RoboDK station: MitsubishiWithPython.rdk

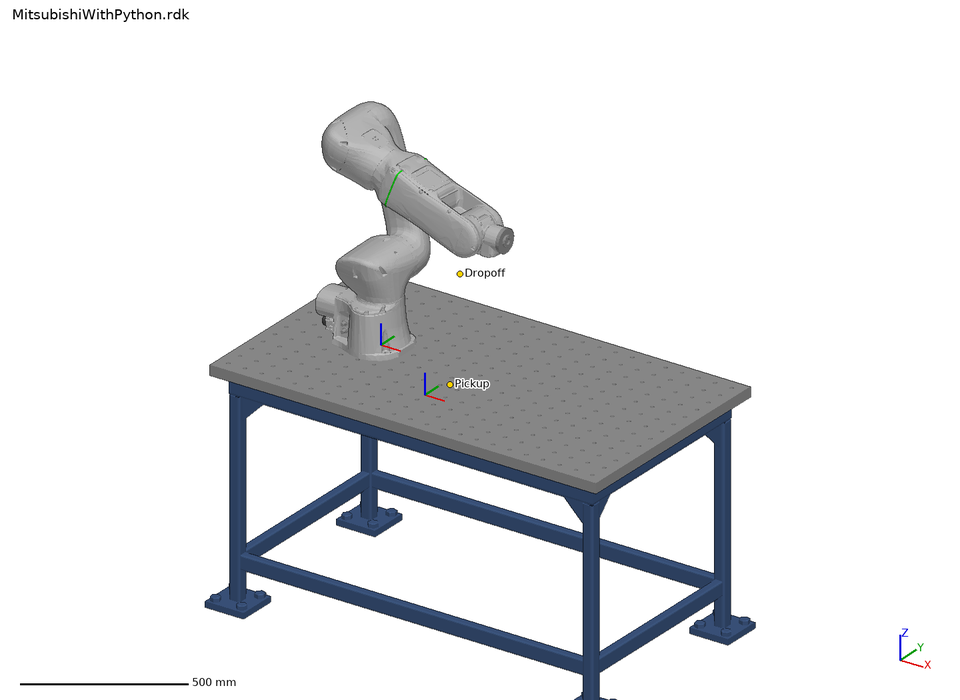
[picture v0: the station drawn from its stored meshes, robots at their saved joint values, targets as dots, program paths as lines]
Station MitsubishiWithPython (saved by RoboDK 5.7.3). Poses are relative to the parent item; angles as X-Y-Z fixed-axis rotations.
  - frame Frame RV-5AS-D at (0, 0, 0) mm
    - robot Mitsubishi RV-5AS-D: 6 axes, payload 5 kg, reach 900 mm, repeatability 0.02 mm, weight 58 kg
        modified DH rows (alpha deg, a mm, theta deg, d mm): 0, 0, 0, 254; -90, 0, -90, 0; 0, 410, -90, 0; -90, 0, 0, 500; 90, 0, 0, 0; -90, 0, 180, 125
        joint limits [-240, -148, -150, -200, -120, -200] to [240, 148, 150, 200, 120, 200]; home [0, 0, 90, 0, 0, 0]; saved at [-1.402, -18.281, 127.838, -4.182, -19.605, 5.574]
  - object Table 1400x800x800mm at (0, 0, 0) mm, size 1420 x 820 x 800 mm, geometry from Table-1400x800x800mm.sld
  - Python program Prog1 (listed below)
  - frame GameFrame at (300, -200, 0) mm
    - target Dropoff (Cartesian target) at (167.45, -58.28, 468.81) mm, rotated rx 90 ry 88.37 rz 90 deg; joints [-37.024, -4.466, 117.289, -62.783, -42.619, 56.684] of Mitsubishi RV-5AS-D
    - target Pickup (Cartesian target) at (71.75, 27.51, 42.52) mm, rotated rx 179.92 ry -4.62 rz -178.08 deg; joints [-24.291, 28.472, 124.985, -183.849, -30.78, 157.175] of Mitsubishi RV-5AS-D

--- Python program Prog1 ---
from robodk.robolink import *  # RoboDK API
from robodk.robomath import *  # RoboDK math utilities

# Initialiser RoboDK API
RDK = Robolink()

# Finn roboten
robot = RDK.Item('', ITEM_TYPE_ROBOT)

if not robot.Valid():
    raise Exception("Ingen robot funnet. Vennligst last inn en robot i RoboDK.")

# Finn targets
pickup_target = RDK.Item("Pickup", ITEM_TYPE_TARGET)
dropoff_target = RDK.Item("Dropoff", ITEM_TYPE_TARGET)

if not pickup_target.Valid() or not dropoff_target.Valid():
    raise Exception("Pickup eller Dropoff target er ikke definert i RoboDK.")

# Flytt roboten til "Pickup"
robot.MoveJ(pickup_target)

# Flytt roboten til "Dropoff"
robot.MoveJ(dropoff_target)

# Startposisjon for offset targets
current_pose = robot.Pose()
for i in range(5):
    # Lag ny posisjon med offset i Y-retning
    offset_pose = current_pose * transl(0, 50 * (i + 1), 0)

    # Flytt roboten til den nye posisjonen
    robot.MoveL(offset_pose)

print("Bevegelse fullført!")
